PROGRAM prgTimeStatistics
VAR
	enableTimeCount: BOOL;
	lastTimeStats:FB_LastTimesStats;
	stats:st_BasicStats;
	lastTime: TIME;
	currTime: TIME;
	lastTimes: ARRAY [1..GVL_Const.lastStatsValue] OF TIME;
	arLastTimes: ARRAY [1..GVL_Const.lastStatsValue] OF LREAL;
END_VAR

lastTimeStats(enable:= enableTimeCount,lastTime => lastTime, currTime=>currTime, lastTimes => lastTimes, arLastTimes => arLastTimes);

stats:=lastTimeStats.M_GetBasicStats();

END_PROGRAM

(* stored: Version 1.1.0.1, ProductVersion 3.1.4024.11
   POU prgTimeStatistics: Id {bbff2c88-80e2-406c-902e-430bf26b8972}, SpecialFunc None *)
